INTERFACE ITF_Receiver EXTENDS __System.IQueryInterface

METHOD flush : BOOL
VAR_INPUT
END_VAR
END_METHOD

METHOD Parse : BOOL
VAR_INPUT
END_VAR
END_METHOD

PROPERTY received : BOOL
GET
END_GET
END_PROPERTY

METHOD ResetBufferPointer : BOOL
VAR_INPUT
END_VAR
END_METHOD

METHOD SetReceivedData : BOOL
VAR_INPUT
	pData	: PVOID;
	cbLen	: UDINT;
END_VAR
END_METHOD

END_INTERFACE

(* stored: Version 1.1.0.1, ProductVersion 3.1.4024.15
   Itf ITF_Receiver: Id {128973b7-40f2-4810-a45e-5d7cb8c99a3f}
   Method flush: Id {74ab21e6-d44b-4e43-8ab5-0213057c280a}
   Method Parse: Id {58faed4d-4787-4aea-a1d8-5f4146bd7808}
   Property received: Id {114c9ed4-9cd8-4d0f-96ef-f0dd65cba216}
   Get Get: Id {d7f3ab06-d17c-4d0c-8428-d71c88069bad}
   Method ResetBufferPointer: Id {38f40fe8-e3b7-4202-b784-5566e03f2db6}
   Method SetReceivedData: Id {296805c3-8e67-4403-b7e7-36f4b85dff67} *)
